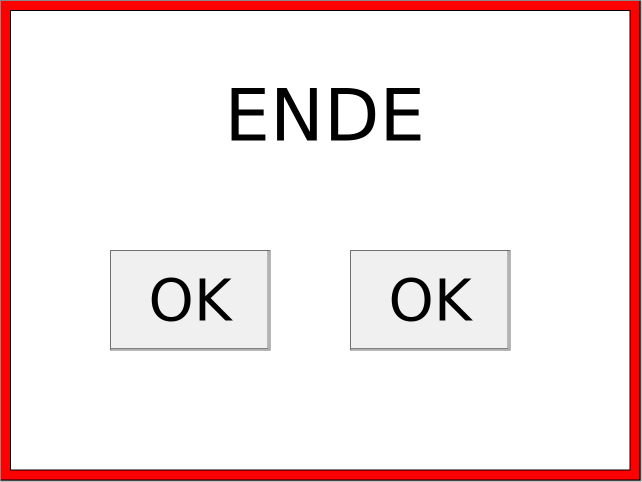
VISUALIZATION Ende  // 642x482
    Rectangle (0,0 640x480)
    Rectangle (10,10 620x460)
    Rectangle (130,50 390x130), "ENDE"
    Button (110,250 160x100), "OK"
        tap MAIN.bOK p1329445385=TRUE
    Button (350,250 160x100), "OK"
        tap MAIN.bOK p1329445385=TRUE
END_VISUALIZATION

(* stored: Version 1.1.0.1, ProductVersion 3.1.4024.0
   Visu Ende: Id {bbd87978-64e2-44d6-bd77-94a7a4e6a086} *)
